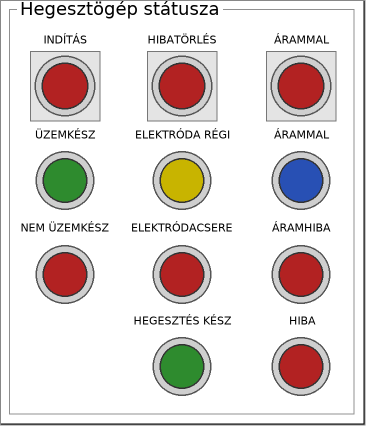
VISUALIZATION Hegeszto_statusz  // 366x426
    Rectangle (0,0 364x424)
    GroupBox (9,1 345x413), "Hegesztögép státusza"
        PushSwitch (138,50 70x70), variable: GVL.bHegesztoHibaTorles, behaviour: TOGGLE, style: Switch-PushSwitch-Red
        PushSwitch (21,50 70x70), variable: HEGESZTOK.bHegesztoStart, behaviour: TOGGLE, style: Switch-PushSwitch-Red
        Label (133,29 80x20), "HIBATÖRLÉS"
        Label (258,29 69x20), "ÁRAMMAL"
        Lamp1 (139,145 68x69), variable: HEGESZTOK.bHegesztoVorwarnung, style: Lamp-Lamp1-Yellow
        Lamp1 (139,239 68x69), variable: HEGESZTOK.bHegesztoElektrodenAnfordem, style: Lamp-Lamp1-Red
        Lamp1 (22,145 68x69), variable: HEGESZTOK.bHegesztoBereit, style: Lamp-Lamp1-Green
        Lamp1 (258,239 68x69), variable: HEGESZTOK.bHegesztoStromFehler, style: Lamp-Lamp1-Red
        Label (258,217 69x20), "ÁRAMHIBA"
        Label (258,124 69x20), "ÁRAMMAL"
        Lamp1 (22,239 68x69), variable: HEGESZTOK.bHegesztoNichtBereit, style: Lamp-Lamp1-Red
        Label (112,124 123x20), "ELEKTRÓDA RÉGI"
        Lamp1 (258,145 68x69), variable: HEGESZTOK.bHegesztoMitStromIn, style: Lamp-Lamp1-Blue
        Label (22,29 69x20), "INDÍTÁS"
        Label (22,124 69x20), "ÜZEMKÉSZ"
        Label (114,217 118x20), "ELEKTRÓDACSERE"
        Label (3,217 106x20), "NEM ÜZEMKÉSZ"
        PushSwitch (257,50 70x70), variable: HEGESZTOK.bHegesztoMitStromOut, behaviour: TOGGLE, style: Switch-PushSwitch-Red
        Lamp1 (258,331 68x69), variable: GVL.bHegesztoHiba, style: Lamp-Lamp1-Red
        Lamp1 (139,331 68x69), variable: HEGESZTOK.bHegesztoFK, style: Lamp-Lamp1-Green
        Label (113,310 121x20), "HEGESZTÉS KÉSZ"
    Label (268,311 69x20), "HIBA"
END_VISUALIZATION

(* stored: Version 1.1.0.1, ProductVersion 3.1.4024.11
   Visu Hegeszto_statusz: Id {bd31292c-dd36-4f61-8315-eb9741e51438} *)
